{attribute 'qualified_only'}
VAR_GLOBAL
	SinOfAngle : LREAL;
END_VAR

(* stored: Version 1.1.0.1, ProductVersion 3.1.4024.12
   GVL GVL: Id {95efe5c4-33b2-4c8a-ac30-e2c3faf0f65c} *)
